INTERFACE I_CTable EXTENDS Debug.I_Debug

PROPERTY Cap : UDINT
GET
END_GET
END_PROPERTY

METHOD Get : Results.Result
VAR_INPUT
	nIndex		: UDINT;
END_VAR
VAR_OUTPUT
	iComponent	: I_Component;
END_VAR
END_METHOD

PROPERTY Length : UDINT
GET
END_GET
END_PROPERTY

END_INTERFACE

(* stored: Version 1.1.0.1
   Itf I_CTable: Id {e42bfe3d-aa88-4aad-be2a-56b20f2b85a6}
   Property Cap: Id {adfe7612-b1e7-4281-ac27-20687e11993a}
   Get Get: Id {92b90c97-ad3f-44e0-ae2c-429f90471f3b}
   Method Get: Id {91c8bc8d-c196-49d9-a3c6-a4f928dfb744}
   Property Length: Id {ebcd1640-4ba5-4382-ba40-ca4aa02566b3}
   Get Get: Id {49e78f87-b82d-4a0b-b831-493ad604eef9} *)
